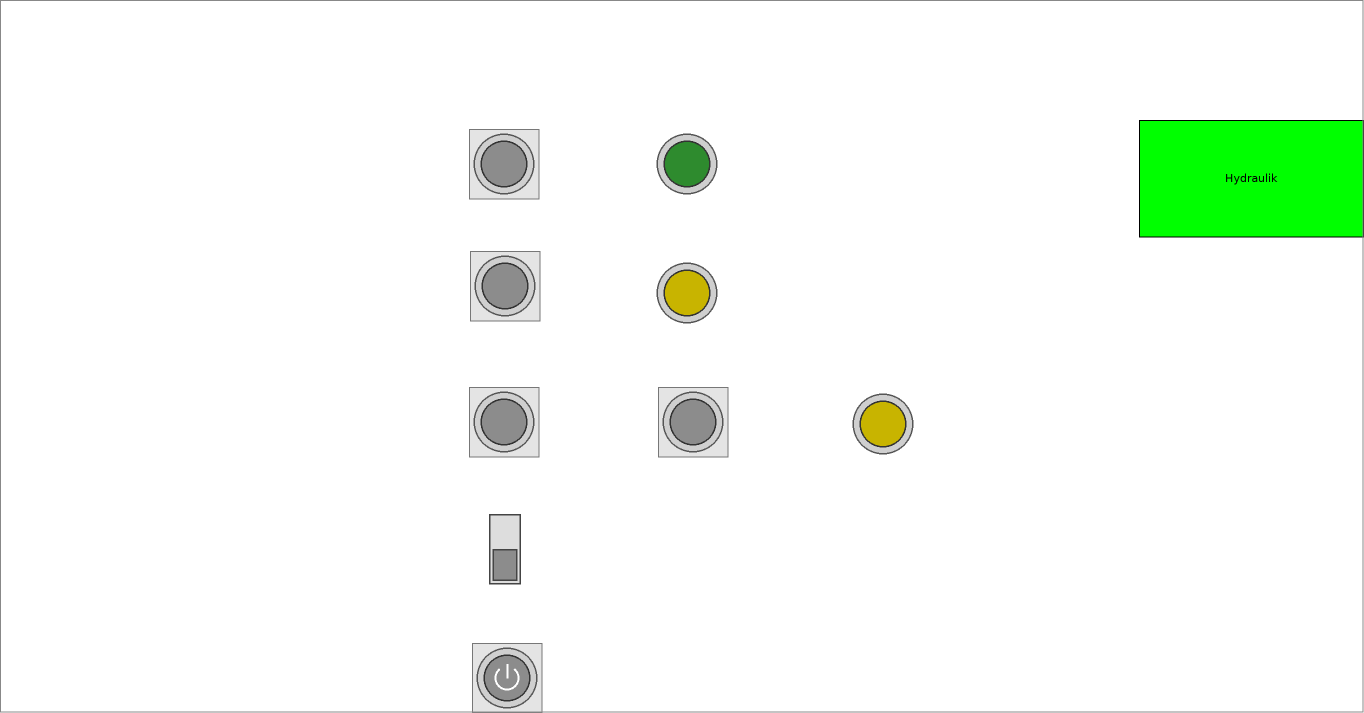
VISUALIZATION Visualization  // 1364x713
    PushSwitch (469,129 70x70), tooltip "Hydraulics start", variable: HydraulicsControl.start, behaviour: TOGGLE, style: Switch-PushSwitch-Gray
    PushSwitch (470,251 70x70), tooltip "Hydraulics stop", variable: HydraulicsControl.stop, behaviour: TOGGLE, style: Switch-PushSwitch-Gray
    Lamp1 (652,129 70x70), tooltip "pump running", variable: HydraulicsControl.pump_running, style: Lamp-Lamp1-Green
    Lamp1 (652,258 70x70), tooltip "suction running", variable: HydraulicsControl.suction_running, style: Lamp-Lamp1-Yellow
    DipSwitch (470,514 70x70), tooltip "Elevation enable", variable: ElevationControl.enable, behaviour: TOGGLE, style: Switch-DipSwitch-Gray
    PushSwitch (658,387 70x70), tooltip "close brake", variable: HydraulicsControl.close_brake, behaviour: TOGGLE, style: Switch-PushSwitch-Gray
    RoundedRectangle (1139,120 225x117), "Hydraulik", colour toggle: HydraulicsControl.pump_running
        tap HydraulicsControl.start
    PowerSwitch (472,643 70x70), variable: TelescopeControl.power, behaviour: TOGGLE, style: Switch-PowerSwitch-Gray
    PushSwitch (469,387 70x70), tooltip "open brake", variable: HydraulicsControl.open_brake, behaviour: TOGGLE, style: Switch-PushSwitch-Gray
    Lamp1 (848,389 70x70), tooltip "brake open", variable: HydraulicsControl.brake_open, style: Lamp-Lamp1-Yellow
END_VISUALIZATION

(* stored: Version 1.1.0.1, ProductVersion 3.1.4024.6
   Visu Visualization: Id {2389e72e-f3ee-4486-a754-3a290b812c2e} *)
